FUNCTION updateDatetimeStamp
VAR_INPUT
	stEvent : REFERENCE TO ST_Event;
	
END_VAR
VAR
	fbgetSystemTime: GETSYSTEMTIME;
	tFilename : T_FILETIME;	
END_VAR

fbgetSystemTime(timeLoDW => tFilename.dwLowDateTime,
	timeHiDW => tFilename.dwHighDateTime);
	
stEvent.dtTimeStamp := FILETIME_TO_DT( filetime:= tFilename);

END_FUNCTION

(* stored: Version 1.1.0.1, ProductVersion 3.1.4024.16
   POU updateDatetimeStamp: Id {461349c2-9e66-4c0d-82de-fe1aef8af1c9}, SpecialFunc None *)
